FUNCTION_BLOCK FB_Conveyor EXTENDS FB_Base IMPLEMENTS I_Device
VAR_INPUT
    bEnable : BOOL;
    rSetSpeed : REAL := 0.0;
END_VAR
VAR_OUTPUT
    bRunning : BOOL;
END_VAR
VAR
    fbMotor : FB_Motor;
    tonDelay : TON;
    eState : E_ConveyorState;
    stConfig : ST_ConveyorConfig;
    _rSpeed : REAL;
END_VAR

tonDelay(IN := bEnable, PT := stConfig.tStartupDelay);
fbMotor(bEnable := bEnable);
bRunning := fbMotor.bActive AND NOT F_IsError(fbMotor);
UpdateState();

METHOD Start : BOOL
VAR_INPUT
    rSpeed : REAL;
END_VAR
IF rSpeed > GVL_Main.rMaxSpeed THEN
    rSpeed := GVL_Main.rMaxSpeed;
END_IF
fbMotor.SetSpeed(rSpeed := rSpeed);
Start := TRUE;
END_METHOD

METHOD PRIVATE UpdateState
CASE eState OF
    E_ConveyorState.Idle:
        IF bEnable THEN
            eState := E_ConveyorState.Starting;
        END_IF
    E_ConveyorState.Starting:
        tonDelay(IN := TRUE, PT := T#500MS);
        IF tonDelay.Q THEN
            eState := E_ConveyorState.Running;
        END_IF
END_CASE
END_METHOD

ACTION A_Reset:
eState := E_ConveyorState.Idle;
bRunning := FALSE;
END_ACTION

PROPERTY Speed : REAL
GET
Speed := _rSpeed;
END_GET
SET
_rSpeed := Speed;
END_SET
END_PROPERTY

END_FUNCTION_BLOCK

(* stored: Version 1.1.0.1, ProductVersion 3.1.4024.12
   POU FB_Conveyor: Id {a1b2c3d4-0001-4000-8000-000000000001}, SpecialFunc None
   Method Start: Id {a1b2c3d4-0002-4000-8000-000000000002}
   Method UpdateState: Id {a1b2c3d4-0003-4000-8000-000000000003}
   Action A_Reset: Id {a1b2c3d4-0004-4000-8000-000000000004}
   Property Speed: Id {a1b2c3d4-0005-4000-8000-000000000005}
   Get Get: Id {a1b2c3d4-0006-4000-8000-000000000006}
   Set Set: Id {a1b2c3d4-0007-4000-8000-000000000007} *)
